FUNCTION_BLOCK FINAL FB_AnalogueOutput EXTENDS FB_EventLogger
VAR_IN_OUT
	Control					: ST_System;
END_VAR
VAR
	_Input					: UINT;					//Raw Input 1 - Analogue
	_Input2					: BOOL;					//Raw Input 2 - Digital
	_ManOnQa				: BOOL;					//Manual On Analogue Input
	_ManQa					: REAL;					//Manual Analogue Input
	_ManOn					: BOOL;					//Manual On
	_ManOff					: BOOL;					//Manual Off
	_ForceOn				: BOOL;					//Force On
	_ForceOff				: BOOL;					//Force Off
	_Fault					: BOOL;					//Fault
	_SimInput				: BOOL;  				//Simulates Analogue Input
	_SimInput2				: BOOL;					//Simulates Digital Input
	_SimInputQa				: REAL;					//Value of Simulated Analogue Input
	_Value_Q	AT %Q*		: BOOL;					//Value of Input - Digital
	_Value_Qa	AT %Q*		: INT;					//Value of Input - Analogue
	_FallingEdge			: BOOL;					//Falling Edge of Value Signal
	_RisingEdge				: BOOL;					//Raising Edge of Value Signal
	_DebounceOn_ET			: REAL;					//Debounce On Elapsed Time
	_DebounceOff_ET			: REAL;					//Debounce Off Elapsed Time
	_FaultTimer_ET			: REAL;					//Fault timer elapsed
	_HighAlarmLimit			: BOOL;					//Input Value is approaching the maximum operating limit.
	_LowAlarmLimit			: BOOL;					//Input Value is approaching the minimum operating limit.
	_HighHighAlarmLimit		: BOOL;					//Input Value is above  the maximum operating limit
	_LowLowAlarmLimit		: BOOL;					//Input Value is below the minimum operating limit.
	_Alarm					: BOOL;					//Device Alarm
	_Warning				: BOOL;					//Device Warning
	_AlarmNum				: DINT;					//Device Alarm Number
	_WarningNum				: DINT;					//Device Warning Number
	_riseEdge				: R_TRIG;				//Rising Edge Value Trigger
	_fallEdge				: F_TRIG;				//Falling Edge Value Trigger
	_ConfInput				: BOOL;					//Confirgured Input
	_DebounceOn_DN			: BOOL;					//Debounce On Timer is Done
	_DebounceOff_DN			: BOOL;					//Debounce Off Timer is Done
	_R_Trig					: ARRAY[0..9] OF R_TRIG;//Private Rising Edge Triggers
END_VAR
VAR PERSISTENT
	_Name					: STRING[15];			//Name for HMI
	_Description			: STRING[40];			//Description for HMI
	_AlarmMute				: BOOL;					//Alarm Mute
	_TypeConfig				: E_AOutputTypeConfig;	//Type congifuration
	_DebounceOn_PT			: REAL;					//Debounce on timer preset time
	_DebounceOff_PT			: REAL;					//Debounce off timer preset time
	_FaultTimer_PT			: REAL;					//Fault timer preset time
	_InputLimitHigh			: REAL;					//HighHigh limit of Raw Input 1
	_InputLimitLow			: REAL;					//Low limit of Raw Input 1
	_InputLimitHighHigh		: REAL;					//HighHigh limit of Raw Input 1
	_InputLimitLowLow		: REAL;					//LowLow limit of Raw Input 1
	_Scale_Qa				: REAL;					//Scale Factor
	_Subtract_Qa			: REAL;					//Subtract a constant from the output
	_Add_Qa					: REAL;					//Add a constant to the output
END_VAR

M_TypeConfig();
M_AlarmMonitor();
M_WarningMonitor();
M_UnlatchManuals();
M_Output();

//Debounce On Timer
IF _ConfInput = TRUE AND NOT _ForceOff AND NOT _ManOff THEN
	_DebounceOn_ET := _DebounceOn_ET + Control.SystemTime.ScanTime;
	_debounceOn_DN := _DebounceOn_ET > _DebounceOn_PT;
ELSE
	_debounceOn_DN := FALSE;
END_IF
IF _debounceOn_DN OR _ForceOn OR _ManOn THEN
	_Value_Q := TRUE;
	_DebounceOff_ET := 0;
END_IF

//Debounce Off Timer
IF _ConfInput = FALSE AND NOT _ForceOn AND NOT _ManOn THEN
	_DebounceOff_ET := _DebounceOff_ET + Control.SystemTime.ScanTime;
	_debounceOff_DN := _DebounceOff_ET > _DebounceOff_PT;
ELSE
	_debounceOff_DN := FALSE;
END_IF
IF _debounceOff_DN OR _ForceOff OR _ManOff THEN
	_Value_Q:= FALSE;
	_DebounceOn_ET := 0;
END_IF

//Rising Edge Trigger 
_riseEdge(CLK := _Value_Q);
_RisingEdge := _riseEdge.Q;

//Falling Edge Trigger
_fallEdge(CLK := _Value_Q);
_FallingEdge := _fallEdge.Q;

{attribute 'monitoring' := 'variable'}
PROPERTY PUBLIC Alarm : Bool
GET
Alarm := _Alarm;
END_GET
END_PROPERTY

{attribute 'monitoring' := 'variable'}
PROPERTY PUBLIC AlarmMute : BOOL
SET
AlarmMute := _AlarmMute;
END_SET
END_PROPERTY

{attribute 'monitoring' := 'variable'}
PROPERTY PUBLIC DebounceOff_ET : real
GET
DebounceOff_ET := _DebounceOff_ET;
END_GET
END_PROPERTY

{attribute 'monitoring' := 'variable'}
PROPERTY PUBLIC DebounceOff_PT : real
GET
DebounceOff_PT := _DebounceOff_PT;
END_GET
SET
_DebounceOff_PT := DebounceOff_PT;
END_SET
END_PROPERTY

{attribute 'monitoring' := 'variable'}
PROPERTY PUBLIC DebounceOn_ET : real
GET
DebounceOn_ET := _DebounceOn_ET;
END_GET
END_PROPERTY

{attribute 'monitoring' := 'variable'}
PROPERTY PUBLIC DebounceOn_PT : real
GET
DebounceOn_PT := _DebounceOn_PT;
END_GET
SET
_DebounceOn_PT := DebounceOn_PT;
END_SET
END_PROPERTY

{attribute 'monitoring' := 'variable'}
PROPERTY PUBLIC Description : String[40]
GET
Description := _Description;
END_GET
SET
_Description := Description;
END_SET
END_PROPERTY

{attribute 'monitoring' := 'variable'}
PROPERTY PUBLIC FallingEdge : Bool
GET
FallingEdge := _FallingEdge;
END_GET
END_PROPERTY

{attribute 'monitoring' := 'variable'}
PROPERTY PUBLIC Fault : Bool
SET
_Fault := Fault;
END_SET
END_PROPERTY

{attribute 'monitoring' := 'variable'}
PROPERTY PUBLIC FaultTimer_ET : real
GET
FaultTimer_ET := _FaultTimer_ET;
END_GET
END_PROPERTY

{attribute 'monitoring' := 'variable'}
PROPERTY PUBLIC FaultTimer_PT : real
GET
FaultTimer_PT := _FaultTimer_PT;
END_GET
SET
_FaultTimer_PT := FaultTimer_PT;
END_SET
END_PROPERTY

{attribute 'monitoring' := 'variable'}
PROPERTY PUBLIC ForceOn : Bool
GET
ForceOn := _ForceOn;
END_GET
SET
_ForceOn := ForceOn;
END_SET
END_PROPERTY

{attribute 'monitoring' := 'variable'}
PROPERTY PUBLIC Input : UINT
GET
Input := _Input;
END_GET
SET // PUBLIC
_Input := Input;
END_SET
END_PROPERTY

{attribute 'monitoring' := 'variable'}
PROPERTY PUBLIC Input2 : Bool
GET
Input2 := _Input2;
END_GET
END_PROPERTY

METHOD PRIVATE M_AlarmMonitor
VAR_INPUT
END_VAR
VAR_INST
END_VAR
VAR_INST // added by the converter: edge detectors and wires of the graphical bodies
    _w1, _w2, _w3, _w4, _w5 : BOOL;
END_VAR
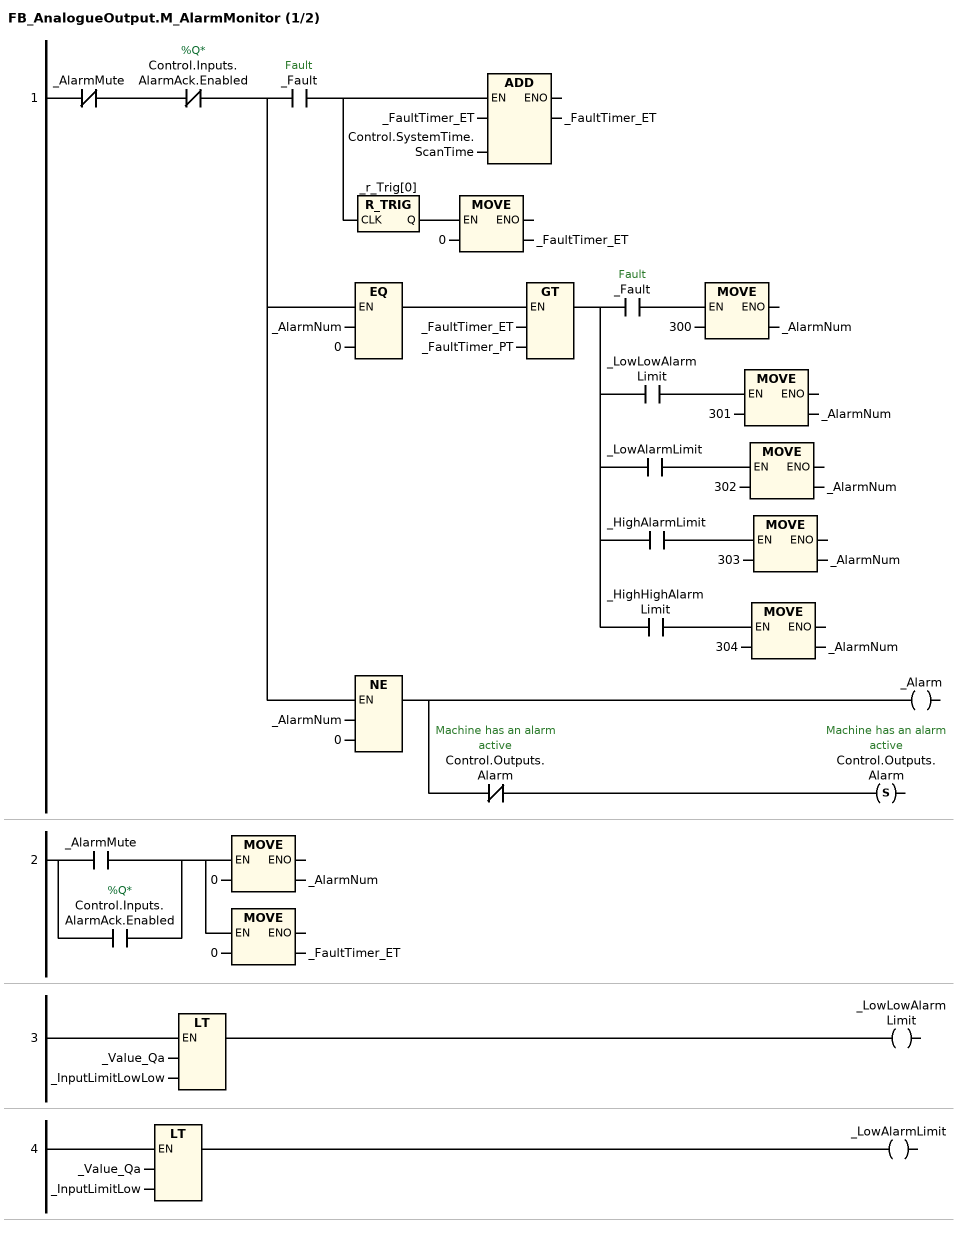
// NETWORK 1
//   Control.Inputs.AlarmAck.Enabled: AT %Q*
//   _Fault: Fault
//   _FaultTimer_ET: Fault timer elapsed
//   Control.SystemTime.ScanTime: Last scan time (Seconds)
//   _FaultTimer_PT: Fault timer preset time
//   Control.Outputs.Alarm: Machine has an alarm active
_w1 := NOT _AlarmMute AND NOT Control.Inputs.AlarmAck.Enabled;
_w2 := _w1 AND _Fault;
IF _w2 THEN _FaultTimer_ET := _FaultTimer_ET + Control.SystemTime.ScanTime; END_IF
_r_Trig[0](CLK := _w2); // R_TRIG
IF _r_Trig[0].Q THEN _FaultTimer_ET := 0; END_IF
_w3 := _w1 AND _AlarmNum = 0 AND _FaultTimer_ET > _FaultTimer_PT;
IF _w3 AND _Fault THEN _AlarmNum := 300; END_IF
IF _w3 AND _LowLowAlarmLimit THEN _AlarmNum := 301; END_IF
IF _w3 AND _LowAlarmLimit THEN _AlarmNum := 302; END_IF
IF _w3 AND _HighAlarmLimit THEN _AlarmNum := 303; END_IF
IF _w3 AND _HighHighAlarmLimit THEN _AlarmNum := 304; END_IF
_w4 := _w1 AND _AlarmNum <> 0;
_Alarm := _w4;
Control.Outputs.Alarm S= _w4 AND NOT Control.Outputs.Alarm;

// NETWORK 2
//   Control.Inputs.AlarmAck.Enabled: AT %Q*
//   _FaultTimer_ET: Fault timer elapsed
_w5 := _AlarmMute OR Control.Inputs.AlarmAck.Enabled;
IF _w5 THEN _AlarmNum := 0; END_IF
IF _w5 THEN _FaultTimer_ET := 0; END_IF

// NETWORK 3
_LowLowAlarmLimit := _Value_Qa < _InputLimitLowLow;

// NETWORK 4
_LowAlarmLimit := _Value_Qa < _InputLimitLow;

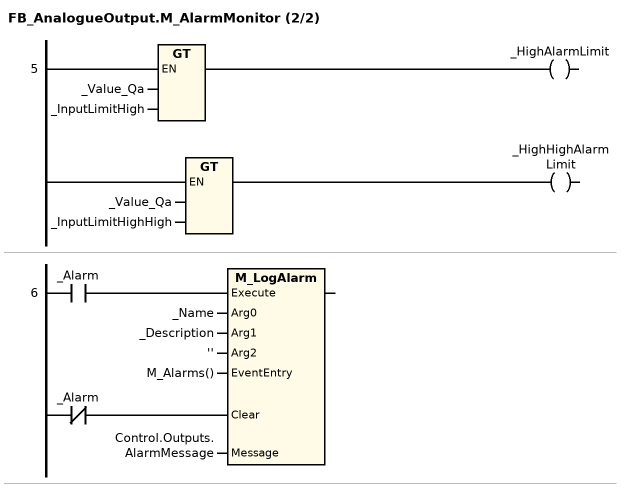
// NETWORK 5
_HighAlarmLimit := _Value_Qa > _InputLimitHigh;
_HighHighAlarmLimit := _Value_Qa > _InputLimitHighHigh;

// NETWORK 6
M_LogAlarm(Execute := _Alarm, Arg0 := _Name, Arg1 := _Description, Arg2 := '', EventEntry := M_Alarms(), Clear := NOT _Alarm, Message := Control.Outputs.AlarmMessage);
END_METHOD

METHOD PRIVATE M_Alarms : TcEventEntry
VAR_INPUT
END_VAR
CASE _AlarmNum OF
	301: M_Alarms:= TC_Events.TcAnalogueOutput.A_301;//Low Low Limit Alarm	
	302: M_Alarms:= TC_Events.TcAnalogueOutput.A_302;//Low Limit Alarm			
	303: M_Alarms:= TC_Events.TcAnalogueOutput.A_303;//High Limit Alarm
	304: M_Alarms:= TC_Events.TcAnalogueOutput.A_304;//High High Limit Alarm							
ELSE
	M_Alarms:= TC_Events.TcAnalogueOutput.A_Undefined;
END_CASE
END_METHOD

METHOD PRIVATE M_Output
VAR_INPUT
END_VAR
VAR_INST
END_VAR
IF _ManOnQa THEN
	IF _Scale_Qa <> 0 THEN
		_Value_Qa :=REAL_TO_INT(_ManQa * _Scale_Qa);
	ELSE
		_Value_Qa :=REAL_TO_INT(_ManQa);
	END_IF	
	
ELSIF _SimInput THEN
	IF _Scale_Qa <> 0 THEN
		_Value_Qa :=REAL_TO_INT(_SimInputQa * _Scale_Qa);
	ELSE
		_Value_Qa :=REAL_TO_INT(_SimInputQa);
	END_IF
	
ELSE
	IF _Scale_Qa <> 0 THEN
		_Value_Qa :=REAL_TO_INT((_Input + _Add_Qa - _Subtract_Qa) * _Scale_Qa);
	ELSE
		_Value_Qa :=REAL_TO_INT( _Input + _Add_Qa - _Subtract_Qa);
	END_IF	
END_IF
END_METHOD

METHOD PRIVATE M_TypeConfig
VAR_INPUT
END_VAR
VAR_INST
END_VAR
CASE _TypeConfig OF
	eAOutputType_PLC_NO, eAOutputType_SAFE_NO : 
		IF _Input2 OR _SimInput2 THEN
			_ConfInput := TRUE;
		ELSE
			_ConfInput := FALSE;
		END_IF
	eAOutputType_PLC_NC, eAOutputType_SAFE_NC : 
		IF NOT _Input2 OR _SimInput2 THEN
			_ConfInput := TRUE;
		ELSE
			_ConfInput := FALSE;
		END_IF
END_CASE
END_METHOD

METHOD PRIVATE M_UnlatchManuals
VAR_INPUT
END_VAR
VAR_INST
END_VAR
VAR_INST // added by the converter: edge detectors and wires of the graphical bodies
    _rt1, _rt2, _rt3 : R_TRIG;
END_VAR
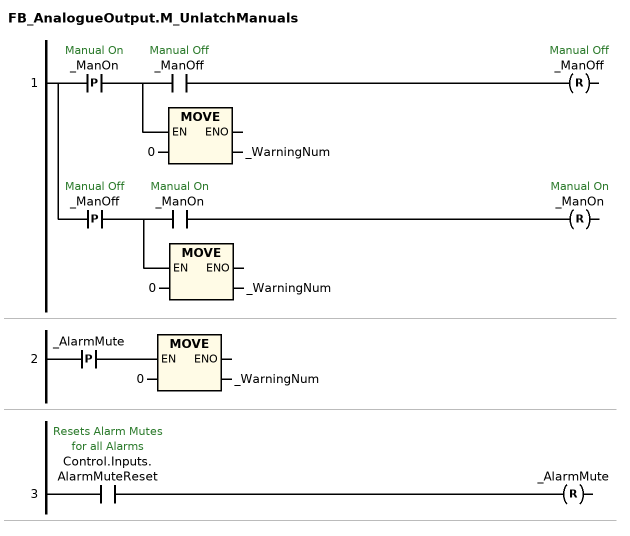
// NETWORK 1
//   _ManOn: Manual On
//   _ManOff: Manual Off
_rt1(CLK := _ManOn);
_ManOff R= _rt1.Q AND _ManOff;
IF _rt1.Q THEN _WarningNum := 0; END_IF
_rt2(CLK := _ManOff);
_ManOn R= _rt2.Q AND _ManOn;
IF _rt2.Q THEN _WarningNum := 0; END_IF

// NETWORK 2
_rt3(CLK := _AlarmMute);
IF _rt3.Q THEN _WarningNum := 0; END_IF

// NETWORK 3
//   Control.Inputs.AlarmMuteReset: Resets Alarm Mutes for all Alarms
_AlarmMute R= Control.Inputs.AlarmMuteReset;
END_METHOD

METHOD PRIVATE M_WarningMonitor
VAR_INPUT
END_VAR
VAR_INST
END_VAR
VAR_INST // added by the converter: edge detectors and wires of the graphical bodies
    _w1 : BOOL;
END_VAR
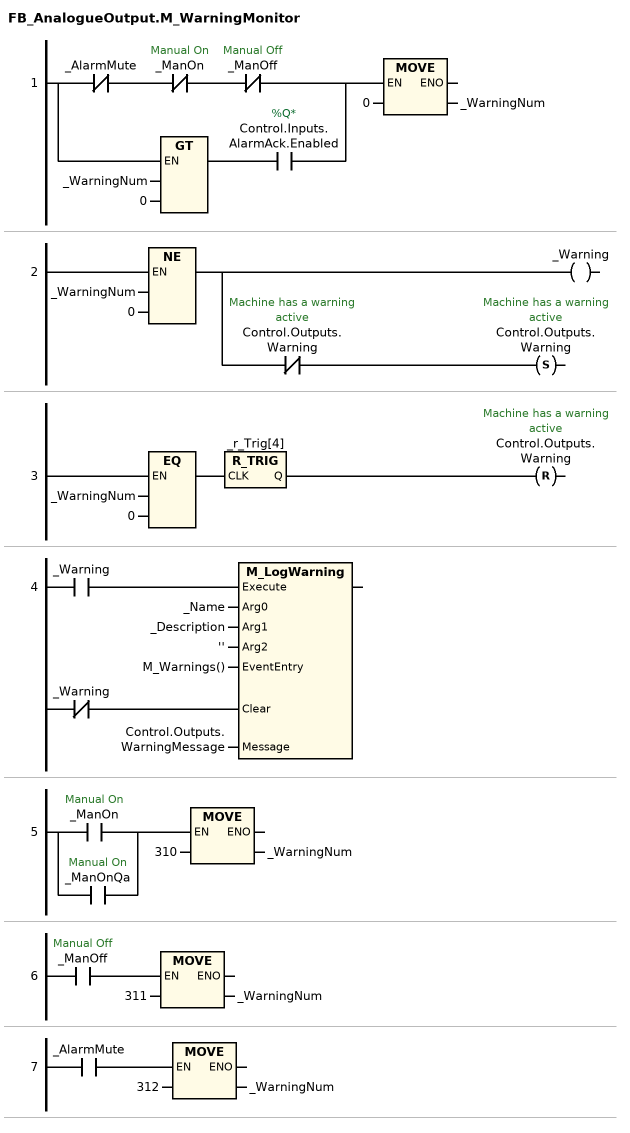
// NETWORK 1
//   _ManOn: Manual On
//   _ManOff: Manual Off
//   Control.Inputs.AlarmAck.Enabled: AT %Q*
IF NOT _AlarmMute AND NOT _ManOn AND NOT _ManOff OR _WarningNum > 0 AND Control.Inputs.AlarmAck.Enabled THEN
    _WarningNum := 0;
END_IF

// NETWORK 2
//   Control.Outputs.Warning: Machine has a warning active
_w1 := _WarningNum <> 0;
_Warning := _w1;
Control.Outputs.Warning S= _w1 AND NOT Control.Outputs.Warning;

// NETWORK 3
//   Control.Outputs.Warning: Machine has a warning active
_r_Trig[4](CLK := _WarningNum = 0); // R_TRIG
Control.Outputs.Warning R= _r_Trig[4].Q;

// NETWORK 4
M_LogWarning(Execute := _Warning, Arg0 := _Name, Arg1 := _Description, Arg2 := '', EventEntry := M_Warnings(), Clear := NOT _Warning, Message := Control.Outputs.WarningMessage);

// NETWORK 5
//   _ManOn: Manual On
//   _ManOnQa: Manual On
IF _ManOn OR _ManOnQa THEN _WarningNum := 310; END_IF

// NETWORK 6
//   _ManOff: Manual Off
IF _ManOff THEN _WarningNum := 311; END_IF

// NETWORK 7
IF _AlarmMute THEN _WarningNum := 312; END_IF
END_METHOD

METHOD PRIVATE M_Warnings : TcEventEntry
VAR_INPUT
END_VAR
CASE _WarningNum OF
	310: M_Warnings:= TC_Events.TcAnalogueOutput.W_310;//Manual ON Enabled	
	311: M_Warnings:= TC_Events.TcAnalogueOutput.W_311;//Manual OFF Enabled			
	312: M_Warnings:= TC_Events.TcAnalogueOutput.W_312;//Alarm Mute Active					
ELSE
	M_Warnings:=  TC_Events.TcAnalogueOutput.W_Undefined;
END_CASE
END_METHOD

{attribute 'monitoring' := 'variable'}
PROPERTY PUBLIC ManOff : Bool
GET
ManOff := _ManOff;
END_GET
SET
_ManOff := ManOff;
END_SET
END_PROPERTY

{attribute 'monitoring' := 'variable'}
PROPERTY PUBLIC ManOn : Bool
GET
ManOn := _ManOn;
END_GET
SET
_ManOn := ManOn;
END_SET
END_PROPERTY

{attribute 'monitoring' := 'variable'}
PROPERTY PUBLIC ManOnQa : Bool
GET
ManOnQa := _ManOnQa;
END_GET
SET
_ManOnQa := ManOnQa;
END_SET
END_PROPERTY

{attribute 'monitoring' := 'variable'}
PROPERTY PUBLIC ManQa : REAL
GET
ManQa := _ManQa;
END_GET
SET
_ManQa := ManQa;
END_SET
END_PROPERTY

{attribute 'monitoring' := 'variable'}
PROPERTY PUBLIC Name : String[15]
GET
Name := _Name;
END_GET
SET
_Name := Name;
END_SET
END_PROPERTY

{attribute 'monitoring' := 'variable'}
PROPERTY PUBLIC RisingEdge : Bool
GET
RisingEdge := _RisingEdge;
END_GET
END_PROPERTY

{attribute 'monitoring' := 'variable'}
PROPERTY PUBLIC SimInput : Bool
SET
_SimInput := SimInput;
END_SET
END_PROPERTY

{attribute 'monitoring' := 'variable'}
PROPERTY PUBLIC SimInput2 : Bool
SET
_SimInput2 := SimInput2;
END_SET
END_PROPERTY

{attribute 'monitoring' := 'variable'}
PROPERTY PUBLIC SimInputQa : REAL
GET
SimInputQa := _SimInputQa;
END_GET
SET
_SimInputQa := SimInputQa;
END_SET
END_PROPERTY

{attribute 'monitoring' := 'variable'}
PROPERTY PUBLIC StandbyReset : Bool
GET
StandbyReset := _ForceOff;
END_GET
SET
_ForceOff := StandbyReset;
END_SET
END_PROPERTY

{attribute 'monitoring' := 'variable'}
PROPERTY PUBLIC Value_Q : BOOL
GET
Value_Q := _Value_Q;
END_GET
SET
_Value_Q := Value_Q;
END_SET
END_PROPERTY

{attribute 'monitoring' := 'variable'}
PROPERTY PUBLIC Value_Qa : INT
GET
Value_Qa := _Value_Qa;
END_GET
SET
_Value_Qa := Value_Qa;
END_SET
END_PROPERTY

{attribute 'monitoring' := 'variable'}
PROPERTY PUBLIC Warning : Bool
GET
Warning := _Warning;
END_GET
END_PROPERTY

END_FUNCTION_BLOCK

(* stored: Version 1.1.0.1, ProductVersion 3.1.4024.3
   POU FB_AnalogueOutput: Id {74edde60-7c9f-4e6f-a804-d140b3d56543}, SpecialFunc None
   Property Alarm: Id {40bd59b6-31c6-4911-92ca-410bf97e64a0}
   Get Get: Id {b2a2a7bc-39ef-4be9-96a6-bc39e3124b65}
   Property AlarmMute: Id {dc6fca9e-f344-44da-8e78-ab87b8fc9e20}
   Set Set: Id {4b2517a5-6a26-45dc-8210-99e2a3317e0f}
   Property DebounceOff_ET: Id {7de0aae2-07d0-4eb2-99a2-04687b72fc85}
   Get Get: Id {3edf4834-2295-4456-adda-28daf3d49938}
   Property DebounceOff_PT: Id {c04a62a3-7952-465e-b4a0-dadc490110ee}
   Get Get: Id {bfa58580-4861-4762-9dee-fa265e05760f}
   Set Set: Id {31429dbf-2db4-4a6f-94e1-bd0c2ec09576}
   Property DebounceOn_ET: Id {565be37f-fd25-4336-91c5-d9fdcd111327}
   Get Get: Id {aa0d9be3-1833-4d26-bd9a-a9f7da5b97b7}
   Property DebounceOn_PT: Id {ea8c7b8f-0136-4e73-8c5a-eff9b7810054}
   Get Get: Id {0770b50e-a494-4051-b116-c97d10369c55}
   Set Set: Id {88937d57-0e97-4b68-b987-4db94bb9ebc0}
   Property Description: Id {b4263c88-7c9a-4781-a922-2d0df571b025}
   Get Get: Id {0dcd696a-bd63-44ff-b627-9f9efd41e715}
   Set Set: Id {7da4fcdd-738a-48a4-8ebb-80a2d207b6ee}
   Property FallingEdge: Id {a43804ef-279c-4af2-a092-d874b2243877}
   Get Get: Id {4182a9bd-7993-42c1-9783-3ebee28f3e73}
   Property Fault: Id {cf72467f-be88-4a5f-8676-165e7fe431e2}
   Set Set: Id {26c62126-4372-4788-9a92-315e4cf80faf}
   Property FaultTimer_ET: Id {8cf9ed59-93e8-4a52-a739-12aee6b6772a}
   Get Get: Id {6285ac6a-5a7b-4075-9a4e-5c178668e468}
   Property FaultTimer_PT: Id {b2d5fd96-4cac-4a9e-9054-cf43fa5701ef}
   Get Get: Id {e652b9ee-458d-4ef4-ba24-923a6a4c2582}
   Set Set: Id {31e2370c-5912-4936-99d2-27d468ab27a3}
   Property ForceOn: Id {a125a4bc-4aec-4696-9b1a-8bcf75b32abf}
   Get Get: Id {411b61b5-cf94-4573-a053-27b08a720436}
   Set Set: Id {941c028e-42a2-4740-9680-b4ef06cfca05}
   Property Input: Id {38c91b26-4cbd-4d82-b3bf-1b89b9aa2140}
   Get Get: Id {a73f88b5-53dd-4fd1-b1d0-58388f68327a}
   Set Set: Id {4a98f2ec-46bf-4807-8a93-e421a94a0adf}
   Property Input2: Id {ec72324f-23e0-4291-9050-5f273ad2f381}
   Get Get: Id {5f5ba78a-ab40-4926-b956-05e90888fea7}
   Method M_AlarmMonitor: Id {0dc016b8-6ad0-4632-be01-5ea50bbc4e16}
   Method M_Alarms: Id {43d35746-f1a6-4ec8-a829-7e90a64865b1}
   Method M_Output: Id {dd54b79a-1491-47a3-a8e9-910ad70c7746}
   Method M_TypeConfig: Id {5bdcdb17-fe9e-4031-bb32-dda755108c38}
   Method M_UnlatchManuals: Id {9cbe3464-61d9-476e-8002-7cc59fa07566}
   Method M_WarningMonitor: Id {d5074f60-77cc-4dff-b440-20a2318705c8}
   Method M_Warnings: Id {56c35a98-781a-4e15-8042-87e87e14ae77}
   Property ManOff: Id {8adefffa-b0a7-4142-bfd9-5a769f45965e}
   Get Get: Id {e169e76c-7ac5-43bf-b7aa-bc0798d1f5d5}
   Set Set: Id {2cc0923a-43e3-44cd-8ebe-c52035043c9a}
   Property ManOn: Id {91679698-6267-4131-94cf-9cfee3dbe3e5}
   Get Get: Id {df5f48f9-c8d9-411e-a912-82792e971ff8}
   Set Set: Id {04ef9dac-9d21-4965-9e55-b3fbf8acbe5f}
   Property ManOnQa: Id {0651b225-d4f1-4c66-8b6c-db2c49a5a1be}
   Get Get: Id {e603d08d-5ead-46e1-9a41-a8ab576d4730}
   Set Set: Id {eacd73fc-e3c7-46b3-8054-5bb3c9711c32}
   Property ManQa: Id {84a276e4-e2b7-4447-bb88-b7bdac2ad2eb}
   Get Get: Id {c5c7caad-dd7b-45e4-a65e-9e3ce0b2d40d}
   Set Set: Id {61d2afee-ba1f-4da2-910c-4e2d68c24759}
   Property Name: Id {7724f18e-4dd4-454e-b926-0ae6d731a69c}
   Get Get: Id {14946d7d-3a88-466b-a1f7-8189d7342a0f}
   Set Set: Id {4eef7e10-aa59-4980-937e-67fdbf9c7b61}
   Property RisingEdge: Id {8197750c-a118-4e33-baa3-5c4d626f4059}
   Get Get: Id {02c8d387-32bf-4136-b20c-6c6fafc720d5}
   Property SimInput: Id {9d4b7f60-d683-4fdb-a41d-c28ba7c0f775}
   Set Set: Id {265e3d30-524d-4a2d-9b40-60fec9ae4536}
   Property SimInput2: Id {d470b727-ca1e-473e-93c9-442ae4afbed2}
   Set Set: Id {41e4aab5-5e55-4311-97c2-adaf04cb5020}
   Property SimInputQa: Id {377135ac-7c12-45e1-9811-0a48af09d315}
   Get Get: Id {a459579d-b538-4f37-a2fe-e317f51d2488}
   Set Set: Id {3faf5de8-a6e8-4b44-85d0-2f06364a2add}
   Property StandbyReset: Id {889a911b-e1d6-4f96-a96e-9ce72b85af08}
   Get Get: Id {72718e2b-0e14-4d12-a056-0cb995916116}
   Set Set: Id {3c69c178-b7b0-4e25-ace9-6571c34a5af9}
   Property Value_Q: Id {467a8610-35b4-45ca-b814-70310acafe0f}
   Get Get: Id {c292f6e3-7731-47c5-82e5-b9f578b8e4f0}
   Set Set: Id {403f6a9f-9b16-4fb3-9813-471b22230b95}
   Property Value_Qa: Id {4944dab6-5b12-460f-a19d-b53698907530}
   Get Get: Id {ea8066ff-967f-4d17-87a9-2a9557bcdb98}
   Set Set: Id {d8f2e44c-af0d-4572-b585-a7e7b6ae9087}
   Property Warning: Id {3f77ec2f-7559-49c1-9333-c8755b13ad8a}
   Get Get: Id {fae93bd3-9201-4060-86d1-4b18a645f4ca} *)
